(* IEC 61131-3 sources: Summary-ETFA22/ahorn/benchmark, 1 file *)

(* ---- weiglTON.st ---- *)
FUNCTION_BLOCK TON

VAR_INPUT
    IN : BOOL;
    PT : UINT;
END_VAR

VAR_OUTPUT
    Q  : BOOL;
    ET : UINT;
END_VAR

IF IN THEN
    Q:= ET = UINT#0;
    IF ET > UINT#0 THEN
        ET := ET - UINT#1;
    ELSE
        ET := UINT#0;
    END_IF
ELSE
    Q  := FALSE;
    ET := PT;
END_IF

END_FUNCTION_BLOCK
